FUNCTION_BLOCK FB_ChooseAction
VAR_INPUT
END_VAR
VAR_OUTPUT
END_VAR
VAR
END_VAR

END_FUNCTION_BLOCK

(* stored: Version 1.1.0.1, ProductVersion 3.1.4022.18
   POU FB_ChooseAction: Id {6e6a5cf2-af70-4f86-924a-c262843e85ff}, SpecialFunc None *)
